FUNCTION_BLOCK ADDFB (* JADE Implementation *)
  (* Standard: 61499-1 *)
  (* Version 1.0, 2015-04-13, Sadik, FraunhoferIGD *)
  (* Compiler header: package fb.rt; *)
  (* Compiler Java Sun JDK 1.5.0 *)
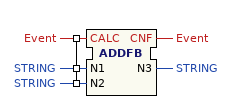
  EVENT_INPUT
    CALC WITH N1, N2; (* Normal Execution Request *)
  END_EVENT
  EVENT_OUTPUT
    CNF; (* Execution Confirmation *)
  END_EVENT
  VAR_INPUT
    N1 : STRING;
    N2 : STRING;
  END_VAR
  VAR_OUTPUT
    N3 : STRING;
  END_VAR
END_FUNCTION_BLOCK
